FUNCTION_BLOCK CM_Actuator3State
VAR_INPUT
	
END_VAR
VAR_OUTPUT
	output_1 : BOOL;
	output_2 : BOOL;
	output_3 : BOOL;
END_VAR
VAR_IN_OUT
	Ctrl_CM_Actuator3State : Udt_CM_Actuator3State;
END_VAR
VAR
END_VAR

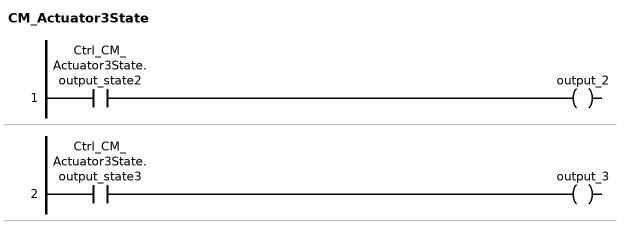
// NETWORK 1
output_2 := Ctrl_CM_Actuator3State.output_state2;

// NETWORK 2
output_3 := Ctrl_CM_Actuator3State.output_state3;

END_FUNCTION_BLOCK

(* stored: Version 1.1.0.1, ProductVersion 3.1.4024.13
   POU CM_Actuator3State: Id {529025ef-40d4-4acc-a1ea-f78f3807d5fa}, SpecialFunc None *)
